(* PLC project Generated.project, CODESYS CODESYS V3.5 SP19 Patch 1 *)
(* stored: creationDateTime 2026-09-06T13:00:42.445772, modificationDateTime 2026-09-06T13:00:42.445772 *)

(* ======================================================================= 🪝 ST_fbWinch_Req — Requête d'axe treuil (producteur PRG_04) ─────────────────────────────────────────────────────────────── 🎯 Rôle : Demande de mouvement, palier et bornes de clamp d'un treuil 📄 Doc métier : DOC/AF/AF_Partie-10_Fonction_Winch_v2.1.md 📤 Producteur : PRG_04_Treuils_Benne (une par treuil M1/M2) 📥 Consommateur : FB_Winch 🔒 Structs cibles + champs conservés pour garder le décodage %→palier et le clamp DANS FB_Winch (comportement bit-identique). SpeedStepReq est consommé par FB_Winch (§5) ; MinStepUp est déclaré mais non consommé (usage aval). ======================================================================= *)
TYPE ST_fbWinch_Req : STRUCT
  RunRequest : BOOL;  (* === ORDRE DE MOUVEMENT === TRUE = mouvement demandé *)
  ReqAscent : BOOL;  (* TRUE = demande montée *)
  ReqDescend : BOOL;  (* TRUE = demande descente *)
  SpeedStepReq : INT;  (* [cible] Palier demandé (1..5, 0 = arrêt) — consommé par FB_Winch *)
  MinStepUp : INT;  (* === BORNES DE CLAMP (agrégées PRG_04) === [cible] Plancher palier montée (usage aval) *)
  MaxStepUp : INT := 5;  (* Plafond palier montée (1..5) *)
  MinStepDown : INT := 0;  (* Plancher palier descente (0 = aucun) -- plongee Kobold *)
  MaxStepDown : INT := 3;  (* Plafond palier descente (1..5) *)
  TopLimitM : REAL := 8.5;  (* === LIMITES EFFECTIVES DU CYCLE === Position limite haute active (m) *)
  BottomLimitM : REAL := -20;  (* Position limite basse active (m) *)
  SyncCoupled : BOOL;  (* === DIAGNOSTIC (jamais lu par la logique FB_Winch) === [diag] Couplage synchro actif (garde de revue) *)
  HomingApproachActive : BOOL;  (* === CHAMPS CONSERVÉS (clamp interne FB_Winch) === [08a] Vitesse limitée au palier 1 (approche homing) *)
END_STRUCT;
END_TYPE
